FUNCTION_BLOCK MSDCmd (* CAT Function Block Type *)
  (* Standard: 61499-2 *)
  (* Version 0.0, 6/7/2026, Schneider Electric, template *)
  PACKAGE SE.Nereda;
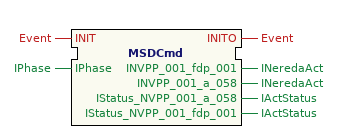
  EVENT_INPUT
    INIT;
  END_EVENT
  EVENT_OUTPUT
    INITO;
  END_EVENT
  SOCKETS
    IPhase : IPhase;
  END_SOCKETS
  PLUGS
    INVPP_001_fdp_001 : INeredaAct;
    INVPP_001_a_058 : INeredaAct;
    IStatus_NVPP_001_a_058 : IActStatus;
    IStatus_NVPP_001_fdp_001 : IActStatus;
  END_PLUGS
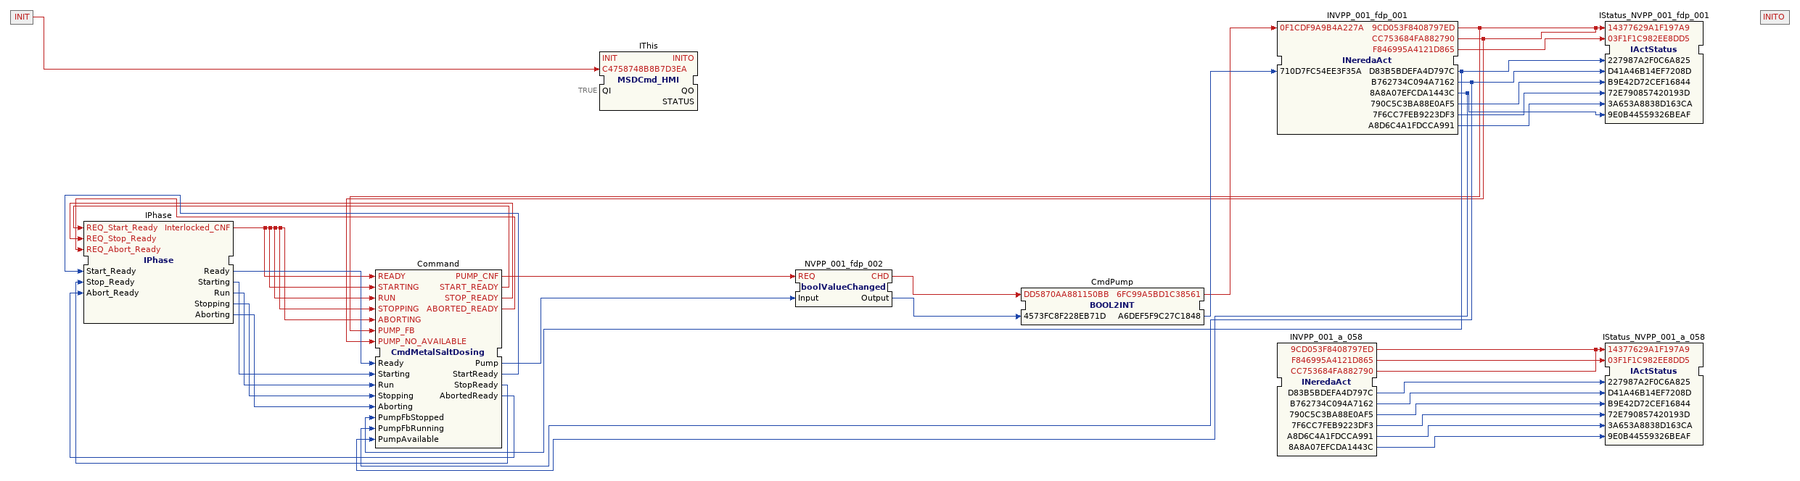
  (* 01 - FUNCTIONNAL INPUT INTERFACE *)
  (* 00 - INITIALIZATION *)
  (* 05 - LOGIC *)
  (* 06 - HMI INTERFACE *)
  (* 03 - FIELD INTERFACE *)
  (* 02 - FUNCTIONNAL OUTPUT INTERFACE *)
  (* Command Logic *)
  FBS
    IThis : MSDCmd_HMI(QI := TRUE);
    Command : CmdMetalSaltDosing;
    NVPP_001_fdp_002 : boolValueChanged;
    CmdPump : BOOL2INT;
  END_FBS
  EVENT_CONNECTIONS
    INIT TO IThis.C4758748B8B7D3EA;
    Command.PUMP_CNF TO NVPP_001_fdp_002.REQ;
    NVPP_001_fdp_002.CHD TO CmdPump.DD5870AA881150BB;
    CmdPump.6FC99A5BD1C38561 TO INVPP_001_fdp_001.0F1CDF9A9B4A227A;
    IPhase.Interlocked_CNF TO Command.READY;
    IPhase.Interlocked_CNF TO Command.STARTING;
    IPhase.Interlocked_CNF TO Command.RUN;
    IPhase.Interlocked_CNF TO Command.STOPPING;
    IPhase.Interlocked_CNF TO Command.ABORTING;
    INVPP_001_fdp_001.9CD053F8408797ED TO Command.PUMP_FB;
    INVPP_001_fdp_001.CC753684FA882790 TO Command.PUMP_NO_AVAILABLE;
    Command.START_READY TO IPhase.REQ_Start_Ready;
    Command.STOP_READY TO IPhase.REQ_Stop_Ready;
    Command.ABORTED_READY TO IPhase.REQ_Abort_Ready;
    INVPP_001_fdp_001.9CD053F8408797ED TO IStatus_NVPP_001_fdp_001.14377629A1F197A9;
    INVPP_001_fdp_001.F846995A4121D865 TO IStatus_NVPP_001_fdp_001.03F1F1C982EE8DD5;
    INVPP_001_a_058.9CD053F8408797ED TO IStatus_NVPP_001_a_058.14377629A1F197A9;
    INVPP_001_a_058.F846995A4121D865 TO IStatus_NVPP_001_a_058.03F1F1C982EE8DD5;
    INVPP_001_fdp_001.CC753684FA882790 TO IStatus_NVPP_001_fdp_001.14377629A1F197A9;
    INVPP_001_a_058.CC753684FA882790 TO IStatus_NVPP_001_a_058.14377629A1F197A9;
  END_CONNECTIONS
  DATA_CONNECTIONS
    Command.Pump TO NVPP_001_fdp_002.Input;
    NVPP_001_fdp_002.Output TO CmdPump.4573FC8F228EB71D;
    CmdPump.A6DEF5F9C27C1848 TO INVPP_001_fdp_001.710D7FC54EE3F35A;
    IPhase.Ready TO Command.Ready;
    IPhase.Starting TO Command.Starting;
    IPhase.Run TO Command.Run;
    IPhase.Stopping TO Command.Stopping;
    IPhase.Aborting TO Command.Aborting;
    INVPP_001_fdp_001.D83B5BDEFA4D797C TO Command.PumpFbStopped;
    INVPP_001_fdp_001.B762734C094A7162 TO Command.PumpFbRunning;
    INVPP_001_fdp_001.8A8A07EFCDA1443C TO Command.PumpAvailable;
    Command.StartReady TO IPhase.Start_Ready;
    Command.StopReady TO IPhase.Stop_Ready;
    Command.AbortedReady TO IPhase.Abort_Ready;
    INVPP_001_fdp_001.D83B5BDEFA4D797C TO IStatus_NVPP_001_fdp_001.227987A2F0C6A825;
    INVPP_001_fdp_001.B762734C094A7162 TO IStatus_NVPP_001_fdp_001.D41A46B14EF7208D;
    INVPP_001_fdp_001.790C5C3BA88E0AF5 TO IStatus_NVPP_001_fdp_001.B9E42D72CEF16844;
    INVPP_001_fdp_001.7F6CC7FEB9223DF3 TO IStatus_NVPP_001_fdp_001.72E790857420193D;
    INVPP_001_fdp_001.A8D6C4A1FDCCA991 TO IStatus_NVPP_001_fdp_001.3A653A8838D163CA;
    INVPP_001_fdp_001.8A8A07EFCDA1443C TO IStatus_NVPP_001_fdp_001.9E0B44559326BEAF;
    INVPP_001_a_058.D83B5BDEFA4D797C TO IStatus_NVPP_001_a_058.227987A2F0C6A825;
    INVPP_001_a_058.B762734C094A7162 TO IStatus_NVPP_001_a_058.D41A46B14EF7208D;
    INVPP_001_a_058.790C5C3BA88E0AF5 TO IStatus_NVPP_001_a_058.B9E42D72CEF16844;
    INVPP_001_a_058.7F6CC7FEB9223DF3 TO IStatus_NVPP_001_a_058.72E790857420193D;
    INVPP_001_a_058.A8D6C4A1FDCCA991 TO IStatus_NVPP_001_a_058.3A653A8838D163CA;
    INVPP_001_a_058.8A8A07EFCDA1443C TO IStatus_NVPP_001_a_058.9E0B44559326BEAF;
  END_CONNECTIONS
END_FUNCTION_BLOCK
